{attribute 'signature_flag' := '1073741824'}
FUNCTION_BLOCK PUBLIC HttpClient
VAR_INPUT
	Execute : BOOL; //REST Call runs on rising edge of this flag 
	Address : STRING(255) := 'https://dog.ceo/api/breeds/image/random'; //Rest API Address
	CallMethod : STRING(255) := 'GET'; //Allowed values are: GET, POST, PUT, DELETE, HEAD, OPTIONS, PATCH, MERGE, COPY.
	Body : STRING(255); //Variable path or string for json body
	ResponseCode : STRING(255); //Variable path to INT for response code
	Response : STRING(255); //Starting variable path to the response
	Port : UINT := 0; //Ads Port for connection. Leave 0 for Port number 851
END_VAR
VAR_OUTPUT
	HasError : BOOL;
	ErrorId : UDINT; //see  ADS error number (https://infosys.beckhoff.com/content/1033/tcplclib_tc2_utilities/45035996647981963.html) or the Win32 error code (https://infosys.beckhoff.com/content/1033/tcplclib_tc2_utilities/27021598155389323.html)
END_VAR
VAR
	startProcess : NT_StartProcess;
	getLocalAmsNetId : FB_GetLocalAmsNetId;
	netIdRead : f_trig;
	initialized : BOOL;
	formatter : FB_FormatString;
END_VAR

startProcess();
getLocalAmsNetId();
startProcess.NETID := getLocalAmsNetId.AddrString;
startProcess.PATHSTR := 'C:\TwinCAT\Functions\Unofficial\BeckhoffHttpClient\TFU001.exe';
startProcess.DIRNAME := 'C:\TwinCAT\Functions\Unofficial\BeckhoffHttpClient\';
formatter(sFormat:='"%s" "%s" "%s" "%s" "%s"', arg1:=f_string(Address), arg2:=f_string(CallMethod), arg3:=f_string(ResponseCode), arg4:=f_string(Body), arg5:=f_string(Response));
IF port <> 0 THEN
	startProcess.COMNDLINE := CONCAT(CONCAT('-AdsPort ',CONCAT(UINT_TO_STRING(Port),' ')),formatter.sOut);
ELSE
	startProcess.COMNDLINE := formatter.sOut;
END_IF

netIdRead(CLK:=getLocalAmsNetId.bBusy, Q=>);

IF netIdRead.Q THEN
	IF NOT getLocalAmsNetId.bError THEN
		initialized := TRUE;
		getLocalAmsNetId.bExecute := FALSE;
	ELSE
		HasError := getLocalAmsNetId.bError;
		ErrorId := getLocalAmsNetId.nErrId;
	END_IF
END_IF

IF NOT initialized THEN
	getLocalAmsNetId.bExecute := TRUE;
END_IF

startProcess.START := initialized AND Execute;

IF initialized THEN
	HasError := startProcess.ERR;
	ErrorId := startProcess.ERRID;
END_IF

END_FUNCTION_BLOCK

(* stored: Version 1.1.0.1, ProductVersion 3.1.4024.3
   POU HttpClient: Id {34d9c780-99db-49b3-b63f-ca9c5a975f9d}, SpecialFunc None *)
